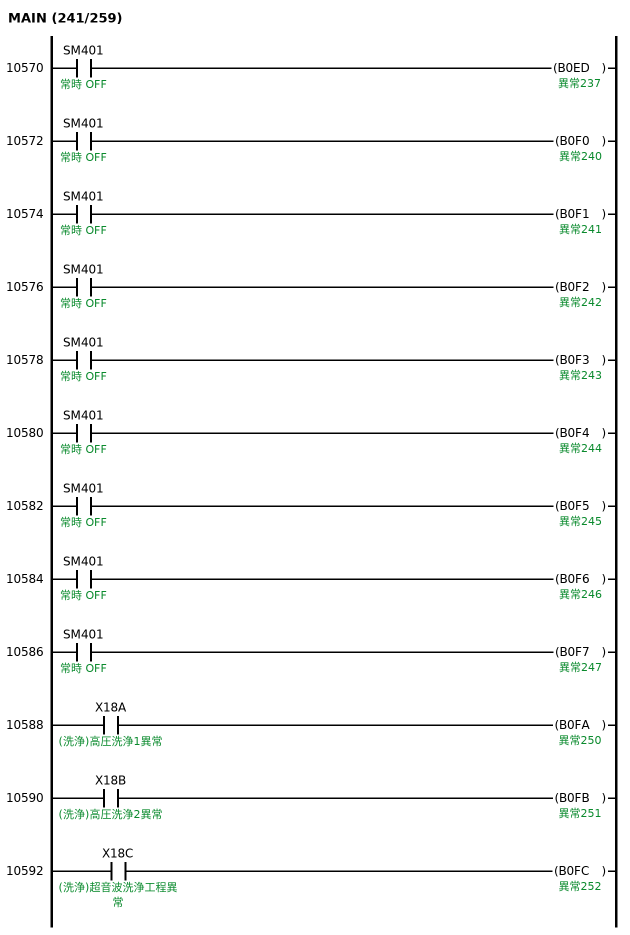
[picture p240: ladder of MAIN, rungs at steps 10570 to 10592]
10570 LD      SM401  ; 常時 OFF
      OUT     B0ED  ; 異常237
10572 LD      SM401  ; 常時 OFF
      OUT     B0F0  ; 異常240
10574 LD      SM401  ; 常時 OFF
      OUT     B0F1  ; 異常241
10576 LD      SM401  ; 常時 OFF
      OUT     B0F2  ; 異常242
10578 LD      SM401  ; 常時 OFF
      OUT     B0F3  ; 異常243
10580 LD      SM401  ; 常時 OFF
      OUT     B0F4  ; 異常244
10582 LD      SM401  ; 常時 OFF
      OUT     B0F5  ; 異常245
10584 LD      SM401  ; 常時 OFF
      OUT     B0F6  ; 異常246
10586 LD      SM401  ; 常時 OFF
      OUT     B0F7  ; 異常247
10588 LD      X18A  ; (洗浄)高圧洗浄1異常
      OUT     B0FA  ; 異常250
10590 LD      X18B  ; (洗浄)高圧洗浄2異常
      OUT     B0FB  ; 異常251
10592 LD      X18C  ; (洗浄)超音波洗浄工程異常
      OUT     B0FC  ; 異常252
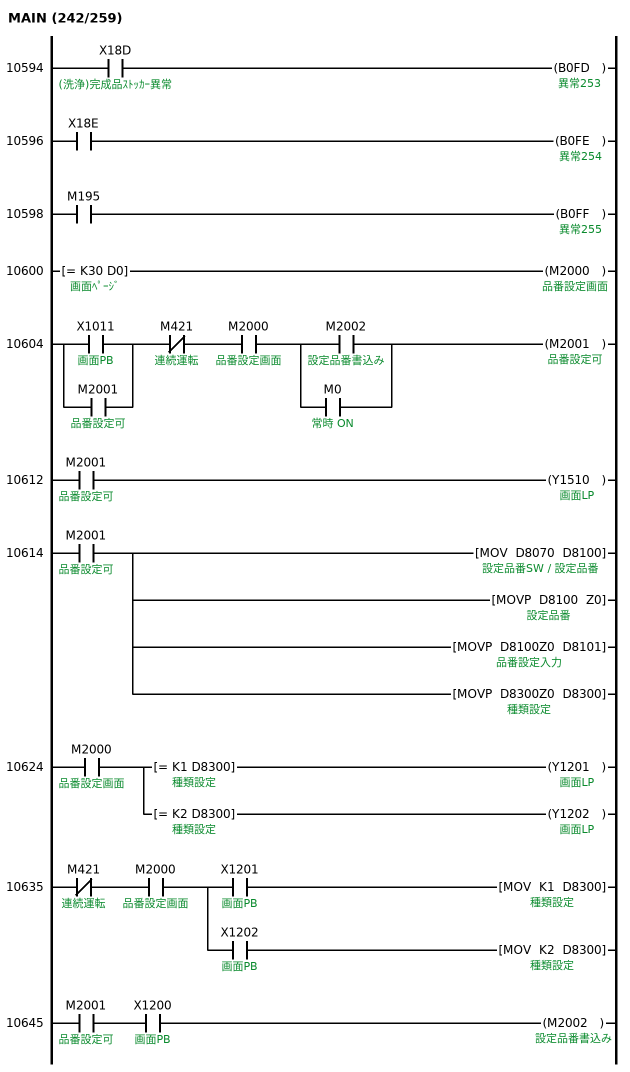
10594 LD      X18D  ; (洗浄)完成品ｽﾄｯｶｰ異常
      OUT     B0FD  ; 異常253
10596 LD      X18E
      OUT     B0FE  ; 異常254
10598 LD      M195
      OUT     B0FF  ; 異常255
10600 LD=     K30 D0  ; 画面ﾍﾟｰｼﾞ
      OUT     M2000  ; 品番設定画面
10604 LD      X1011  ; 画面PB
      OR      M2001  ; 品番設定可
      ANI     M421  ; 連続運転
      AND     M2000  ; 品番設定画面
      LD      M2002  ; 設定品番書込み
      OR      M0  ; 常時 ON
      ANB
      OUT     M2001  ; 品番設定可
10612 LD      M2001  ; 品番設定可
      OUT     Y1510  ; 画面LP
10614 LD      M2001  ; 品番設定可
      MOV     D8070 D8100  ; 設定品番SW / 設定品番
      MOVP    D8100 Z0
      MOVP    D8100Z0 D8101  ; 品番設定入力
      MOVP    D8300Z0 D8300
10624 LD      M2000  ; 品番設定画面
      MPS
      AND=    K1 D8300  ; 種類設定
      OUT     Y1201  ; 画面LP
      MPP
      AND=    K2 D8300  ; 種類設定
      OUT     Y1202  ; 画面LP
10635 LDI     M421  ; 連続運転
      AND     M2000  ; 品番設定画面
      MPS
      AND     X1201  ; 画面PB
      MOV     K1 D8300
      MPP
      AND     X1202  ; 画面PB
      MOV     K2 D8300
10645 LD      M2001  ; 品番設定可
      AND     X1200  ; 画面PB
      OUT     M2002  ; 設定品番書込み
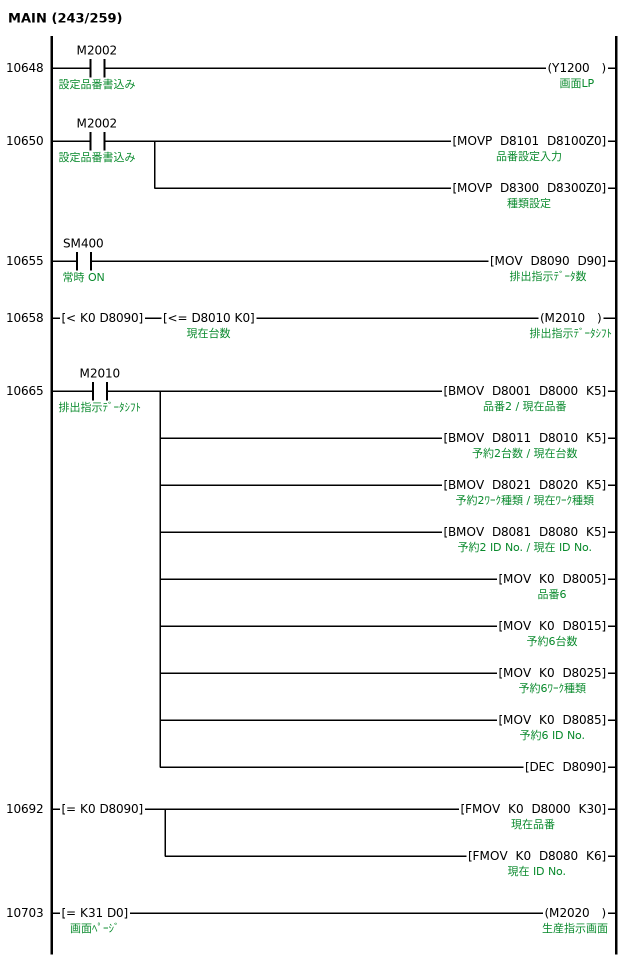
10648 LD      M2002  ; 設定品番書込み
      OUT     Y1200  ; 画面LP
10650 LD      M2002  ; 設定品番書込み
      MOVP    D8101 D8100Z0
      MOVP    D8300 D8300Z0
10655 LD      SM400  ; 常時 ON
      MOV     D8090 D90  ; 排出指示ﾃﾞｰﾀ数
10658 LD<     K0 D8090
      AND<=   D8010 K0  ; 現在台数
      OUT     M2010  ; 排出指示ﾃﾞｰﾀｼﾌﾄ
10665 LD      M2010  ; 排出指示ﾃﾞｰﾀｼﾌﾄ
      BMOV    D8001 D8000 K5  ; 品番2
      BMOV    D8011 D8010 K5  ; 予約2台数
      BMOV    D8021 D8020 K5  ; 予約2ﾜｰｸ種類 / 現在ﾜｰｸ種類
      BMOV    D8081 D8080 K5  ; 予約2 ID No. / 現在 ID No.
      MOV     K0 D8005  ; 品番6
      MOV     K0 D8015  ; 予約6台数
      MOV     K0 D8025  ; 予約6ﾜｰｸ種類
      MOV     K0 D8085  ; 予約6 ID No.
      DEC     D8090
10692 LD=     K0 D8090
      FMOV    K0 D8000 K30
      FMOV    K0 D8080 K6
10703 LD=     K31 D0  ; 画面ﾍﾟｰｼﾞ
      OUT     M2020  ; 生産指示画面
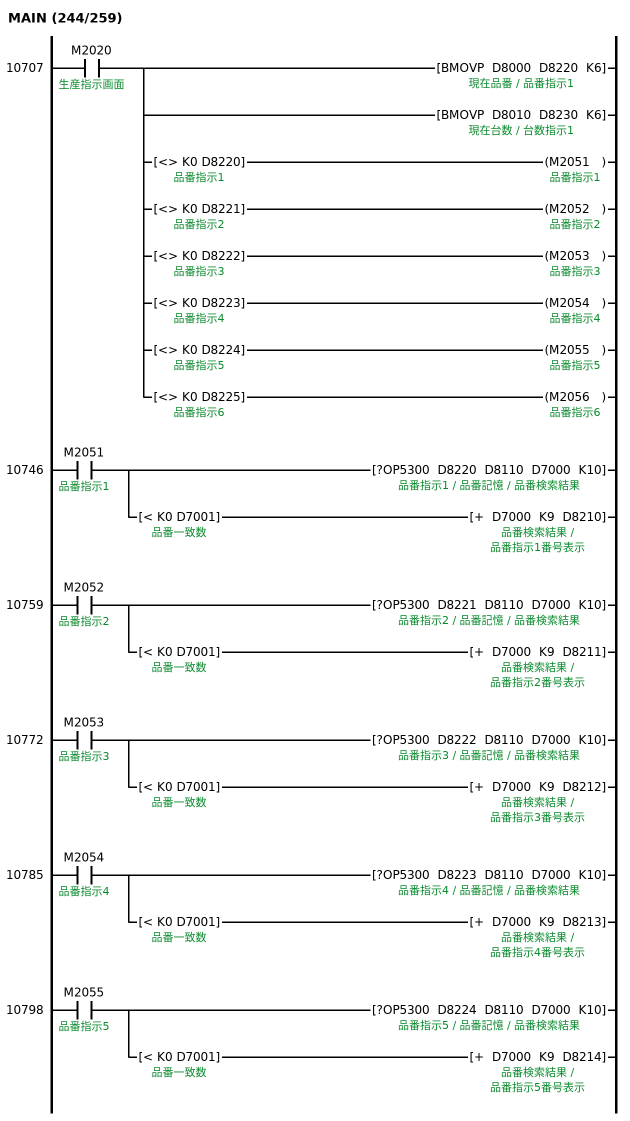
10707 LD      M2020  ; 生産指示画面
      BMOVP   D8000 D8220 K6  ; 品番指示1
      BMOVP   D8010 D8230 K6  ; 台数指示1
      MPS
      AND<>   K0 D8220  ; 品番指示1
      OUT     M2051  ; 品番指示1
      MRD
      AND<>   K0 D8221  ; 品番指示2
      OUT     M2052  ; 品番指示2
      MRD
      AND<>   K0 D8222  ; 品番指示3
      OUT     M2053  ; 品番指示3
      MRD
      AND<>   K0 D8223  ; 品番指示4
      OUT     M2054  ; 品番指示4
      MRD
      AND<>   K0 D8224  ; 品番指示5
      OUT     M2055  ; 品番指示5
      MPP
      AND<>   K0 D8225  ; 品番指示6
      OUT     M2056  ; 品番指示6
10746 LD      M2051  ; 品番指示1
      ?OP5300 D8220 D8110 D7000 K10  ; 品番記憶 / 品番検索結果
      AND<    K0 D7001  ; 品番一致数
      +       D7000 K9 D8210  ; 品番指示1番号表示
10759 LD      M2052  ; 品番指示2
      ?OP5300 D8221 D8110 D7000 K10
      AND<    K0 D7001  ; 品番一致数
      +       D7000 K9 D8211  ; 品番指示2番号表示
10772 LD      M2053  ; 品番指示3
      ?OP5300 D8222 D8110 D7000 K10
      AND<    K0 D7001  ; 品番一致数
      +       D7000 K9 D8212  ; 品番指示3番号表示
10785 LD      M2054  ; 品番指示4
      ?OP5300 D8223 D8110 D7000 K10
      AND<    K0 D7001  ; 品番一致数
      +       D7000 K9 D8213  ; 品番指示4番号表示
10798 LD      M2055  ; 品番指示5
      ?OP5300 D8224 D8110 D7000 K10
      AND<    K0 D7001  ; 品番一致数
      +       D7000 K9 D8214  ; 品番指示5番号表示
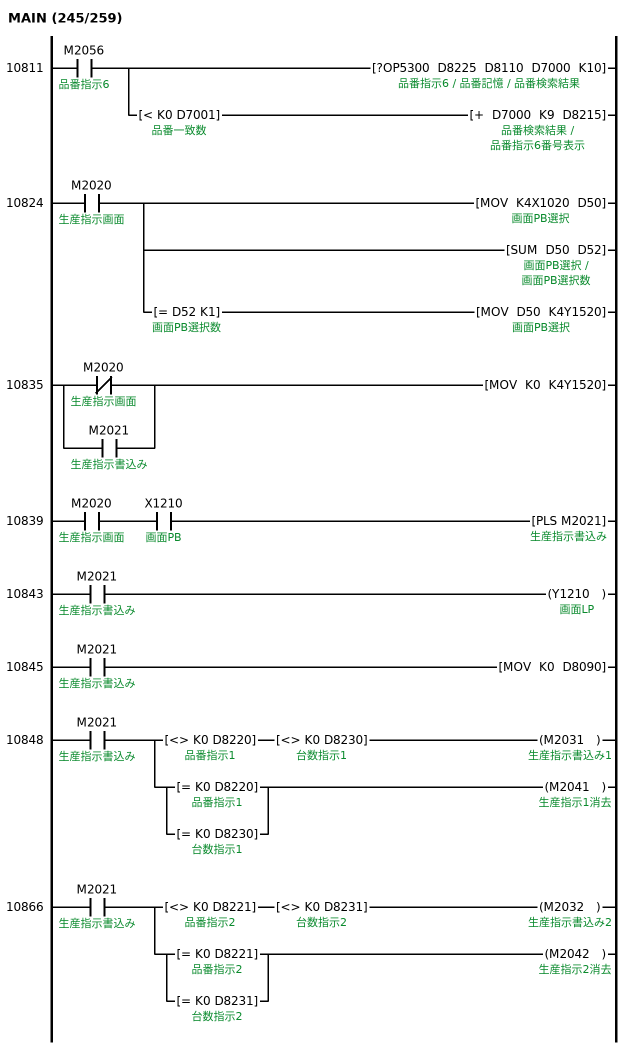
10811 LD      M2056  ; 品番指示6
      ?OP5300 D8225 D8110 D7000 K10
      AND<    K0 D7001  ; 品番一致数
      +       D7000 K9 D8215  ; 品番指示6番号表示
10824 LD      M2020  ; 生産指示画面
      MOV     K4X1020 D50  ; 画面PB
      SUM     D50 D52
      AND=    D52 K1  ; 画面PB選択数
      MOV     D50 K4Y1520  ; 画面LP
10835 LDI     M2020  ; 生産指示画面
      OR      M2021  ; 生産指示書込み
      MOV     K0 K4Y1520
10839 LD      M2020  ; 生産指示画面
      AND     X1210  ; 画面PB
      PLS     M2021  ; 生産指示書込み
10843 LD      M2021  ; 生産指示書込み
      OUT     Y1210  ; 画面LP
10845 LD      M2021  ; 生産指示書込み
      MOV     K0 D8090
10848 LD      M2021  ; 生産指示書込み
      MPS
      AND<>   K0 D8220  ; 品番指示1
      AND<>   K0 D8230  ; 台数指示1
      OUT     M2031  ; 生産指示書込み1
      MPP
      LD=     K0 D8220  ; 品番指示1
      OR=     K0 D8230  ; 台数指示1
      ANB
      OUT     M2041  ; 生産指示1消去
10866 LD      M2021  ; 生産指示書込み
      MPS
      AND<>   K0 D8221  ; 品番指示2
      AND<>   K0 D8231  ; 台数指示2
      OUT     M2032  ; 生産指示書込み2
      MPP
      LD=     K0 D8221  ; 品番指示2
      OR=     K0 D8231  ; 台数指示2
      ANB
      OUT     M2042  ; 生産指示2消去
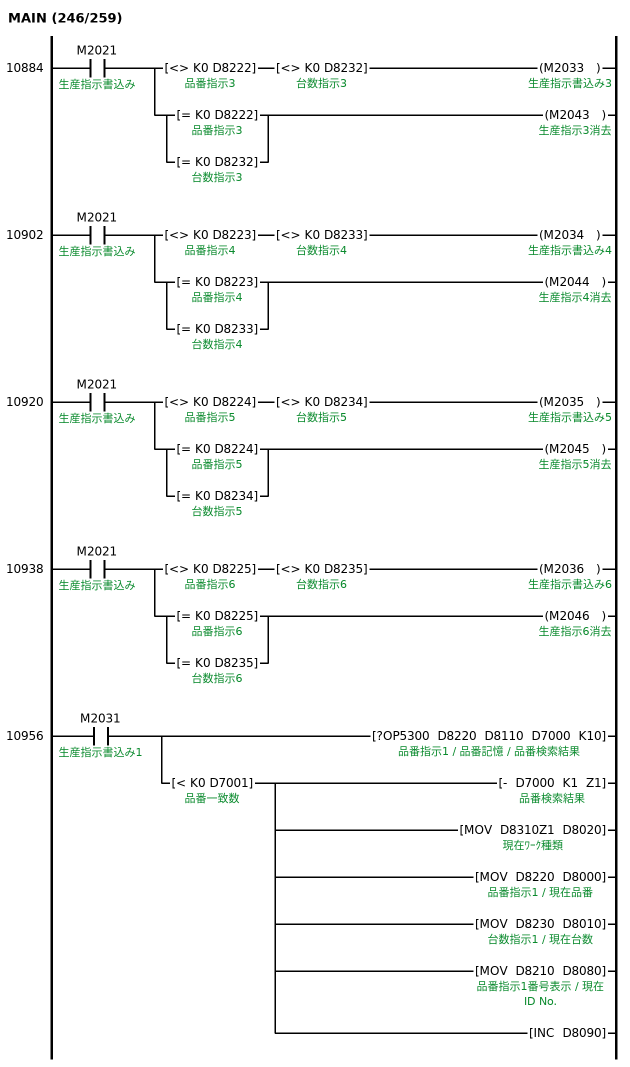
10884 LD      M2021  ; 生産指示書込み
      MPS
      AND<>   K0 D8222  ; 品番指示3
      AND<>   K0 D8232  ; 台数指示3
      OUT     M2033  ; 生産指示書込み3
      MPP
      LD=     K0 D8222  ; 品番指示3
      OR=     K0 D8232  ; 台数指示3
      ANB
      OUT     M2043  ; 生産指示3消去
10902 LD      M2021  ; 生産指示書込み
      MPS
      AND<>   K0 D8223  ; 品番指示4
      AND<>   K0 D8233  ; 台数指示4
      OUT     M2034  ; 生産指示書込み4
      MPP
      LD=     K0 D8223  ; 品番指示4
      OR=     K0 D8233  ; 台数指示4
      ANB
      OUT     M2044  ; 生産指示4消去
10920 LD      M2021  ; 生産指示書込み
      MPS
      AND<>   K0 D8224  ; 品番指示5
      AND<>   K0 D8234  ; 台数指示5
      OUT     M2035  ; 生産指示書込み5
      MPP
      LD=     K0 D8224  ; 品番指示5
      OR=     K0 D8234  ; 台数指示5
      ANB
      OUT     M2045  ; 生産指示5消去
10938 LD      M2021  ; 生産指示書込み
      MPS
      AND<>   K0 D8225  ; 品番指示6
      AND<>   K0 D8235  ; 台数指示6
      OUT     M2036  ; 生産指示書込み6
      MPP
      LD=     K0 D8225  ; 品番指示6
      OR=     K0 D8235  ; 台数指示6
      ANB
      OUT     M2046  ; 生産指示6消去
10956 LD      M2031  ; 生産指示書込み1
      ?OP5300 D8220 D8110 D7000 K10
      AND<    K0 D7001  ; 品番一致数
      -       D7000 K1 Z1
      MOV     D8310Z1 D8020
      MOV     D8220 D8000
      MOV     D8230 D8010
      MOV     D8210 D8080
      INC     D8090
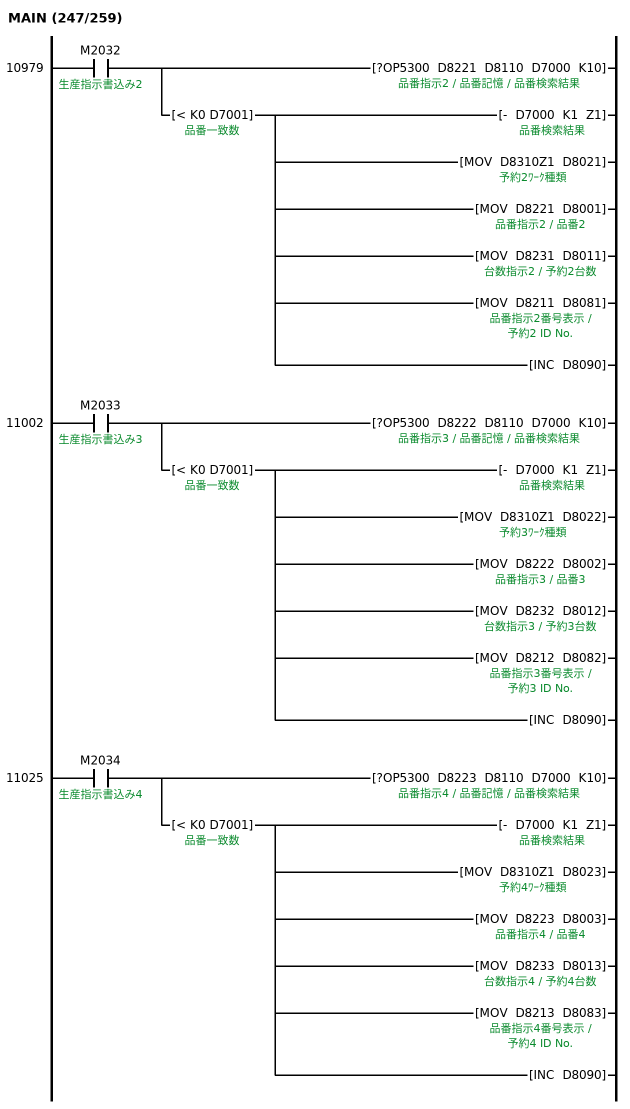
10979 LD      M2032  ; 生産指示書込み2
      ?OP5300 D8221 D8110 D7000 K10
      AND<    K0 D7001  ; 品番一致数
      -       D7000 K1 Z1
      MOV     D8310Z1 D8021
      MOV     D8221 D8001
      MOV     D8231 D8011
      MOV     D8211 D8081
      INC     D8090
11002 LD      M2033  ; 生産指示書込み3
      ?OP5300 D8222 D8110 D7000 K10
      AND<    K0 D7001  ; 品番一致数
      -       D7000 K1 Z1
      MOV     D8310Z1 D8022  ; 予約3ﾜｰｸ種類
      MOV     D8222 D8002  ; 品番3
      MOV     D8232 D8012  ; 予約3台数
      MOV     D8212 D8082  ; 予約3 ID No.
      INC     D8090
11025 LD      M2034  ; 生産指示書込み4
      ?OP5300 D8223 D8110 D7000 K10
      AND<    K0 D7001  ; 品番一致数
      -       D7000 K1 Z1
      MOV     D8310Z1 D8023  ; 予約4ﾜｰｸ種類
      MOV     D8223 D8003  ; 品番4
      MOV     D8233 D8013  ; 予約4台数
      MOV     D8213 D8083  ; 予約4 ID No.
      INC     D8090
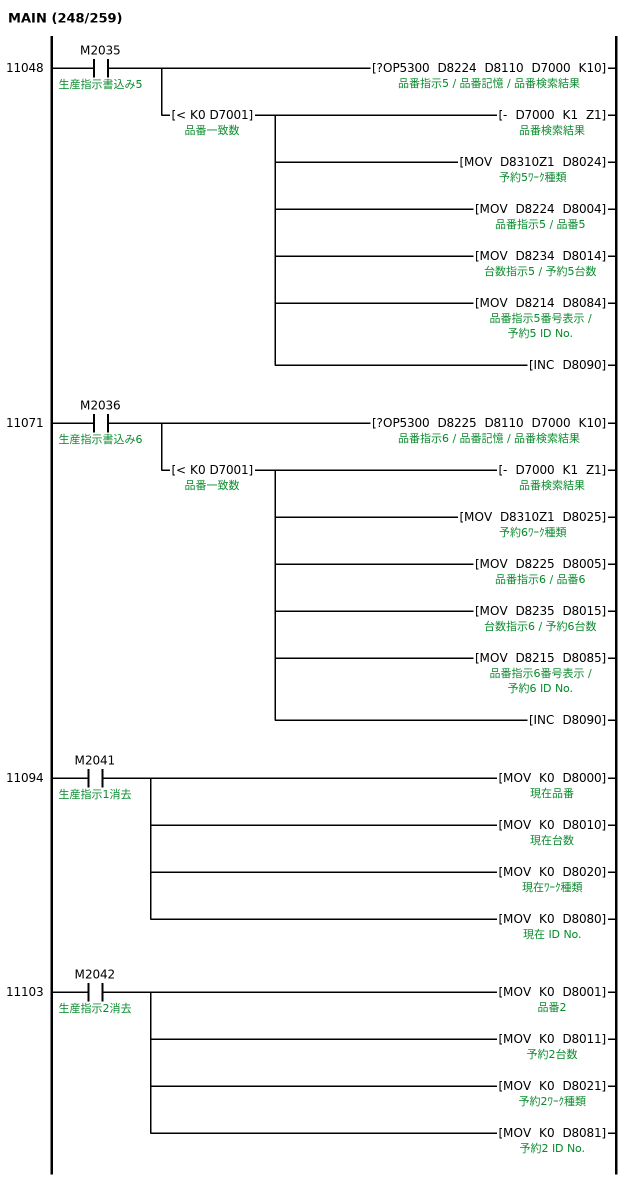
11048 LD      M2035  ; 生産指示書込み5
      ?OP5300 D8224 D8110 D7000 K10
      AND<    K0 D7001  ; 品番一致数
      -       D7000 K1 Z1
      MOV     D8310Z1 D8024  ; 予約5ﾜｰｸ種類
      MOV     D8224 D8004  ; 品番5
      MOV     D8234 D8014  ; 予約5台数
      MOV     D8214 D8084  ; 予約5 ID No.
      INC     D8090
11071 LD      M2036  ; 生産指示書込み6
      ?OP5300 D8225 D8110 D7000 K10
      AND<    K0 D7001  ; 品番一致数
      -       D7000 K1 Z1
      MOV     D8310Z1 D8025
      MOV     D8225 D8005
      MOV     D8235 D8015
      MOV     D8215 D8085
      INC     D8090
11094 LD      M2041  ; 生産指示1消去
      MOV     K0 D8000
      MOV     K0 D8010
      MOV     K0 D8020
      MOV     K0 D8080
11103 LD      M2042  ; 生産指示2消去
      MOV     K0 D8001
      MOV     K0 D8011
      MOV     K0 D8021
      MOV     K0 D8081
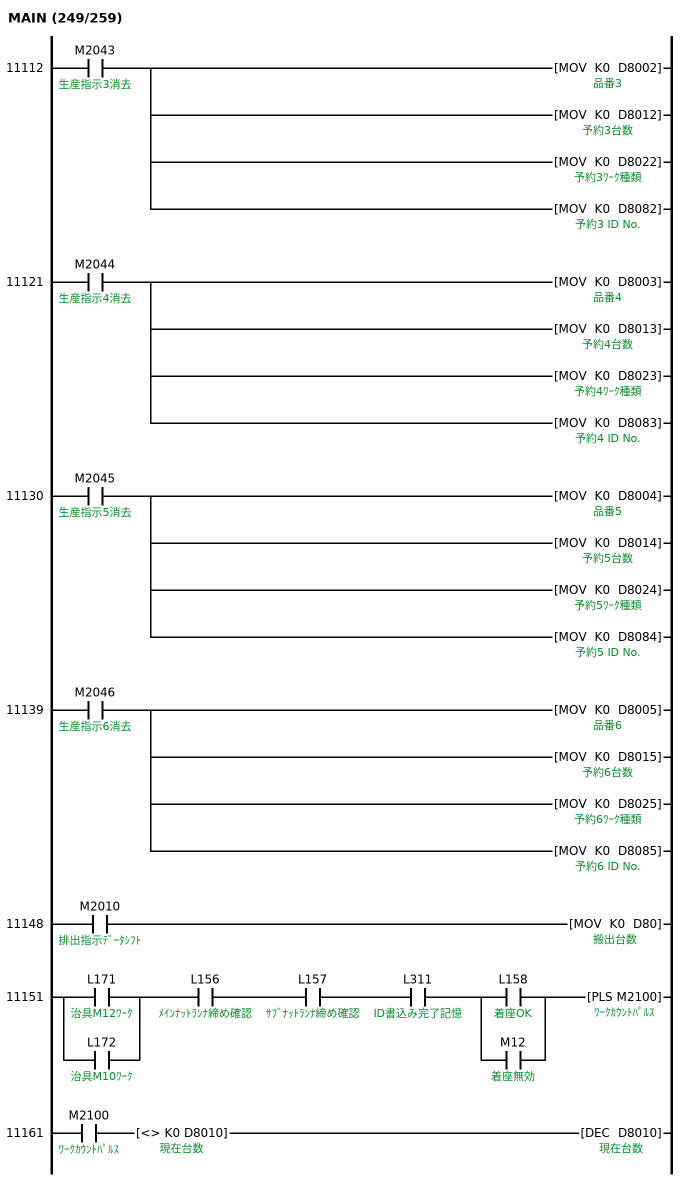
11112 LD      M2043  ; 生産指示3消去
      MOV     K0 D8002
      MOV     K0 D8012
      MOV     K0 D8022
      MOV     K0 D8082
11121 LD      M2044  ; 生産指示4消去
      MOV     K0 D8003
      MOV     K0 D8013
      MOV     K0 D8023
      MOV     K0 D8083
11130 LD      M2045  ; 生産指示5消去
      MOV     K0 D8004
      MOV     K0 D8014
      MOV     K0 D8024
      MOV     K0 D8084
11139 LD      M2046  ; 生産指示6消去
      MOV     K0 D8005
      MOV     K0 D8015
      MOV     K0 D8025
      MOV     K0 D8085
11148 LD      M2010  ; 排出指示ﾃﾞｰﾀｼﾌﾄ
      MOV     K0 D80  ; 搬出台数
11151 LD      L171  ; 治具M12ﾜｰｸ
      OR      L172  ; 治具M10ﾜｰｸ
      AND     L156  ; ﾒｲﾝﾅｯﾄﾗﾝﾅ締め確認
      AND     L157  ; ｻﾌﾞﾅｯﾄﾗﾝﾅ締め確認
      AND     L311  ; ID書込み完了記憶
      LD      L158  ; 着座OK
      OR      M12  ; 着座無効
      ANB
      PLS     M2100  ; ﾜｰｸｶｳﾝﾄﾊﾟﾙｽ
11161 LD      M2100  ; ﾜｰｸｶｳﾝﾄﾊﾟﾙｽ
      AND<>   K0 D8010  ; 現在台数
      DEC     D8010
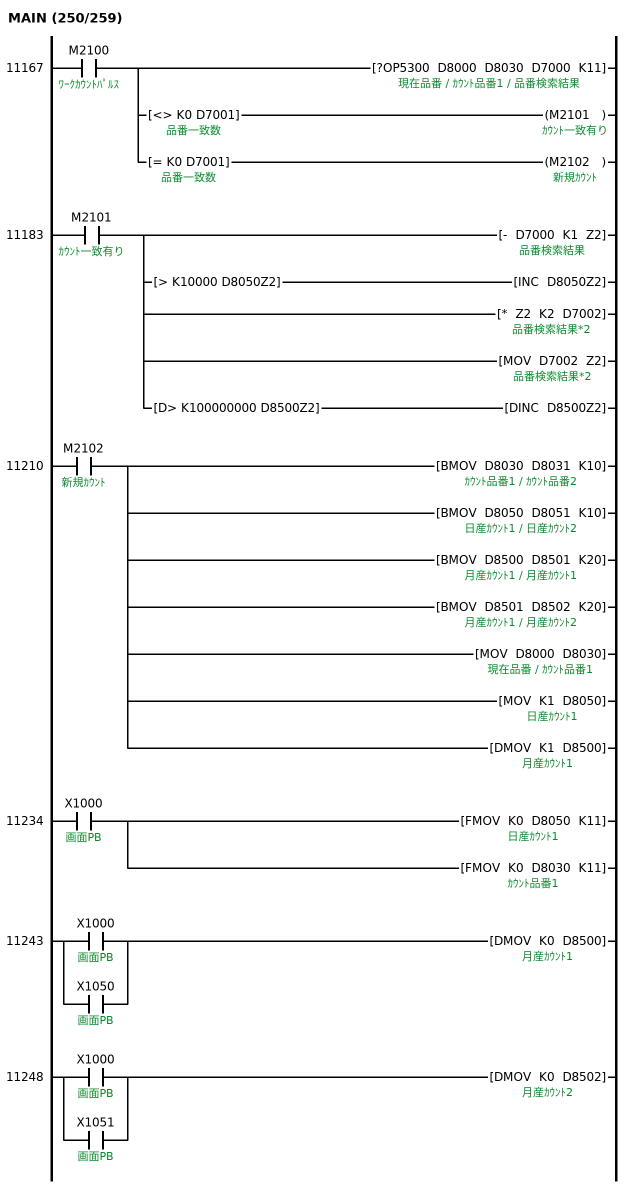
11167 LD      M2100  ; ﾜｰｸｶｳﾝﾄﾊﾟﾙｽ
      ?OP5300 D8000 D8030 D7000 K11  ; ｶｳﾝﾄ品番1
      MPS
      AND<>   K0 D7001  ; 品番一致数
      OUT     M2101  ; ｶｳﾝﾄ一致有り
      MPP
      AND=    K0 D7001  ; 品番一致数
      OUT     M2102  ; 新規ｶｳﾝﾄ
11183 LD      M2101  ; ｶｳﾝﾄ一致有り
      -       D7000 K1 Z2
      MPS
      AND>    K10000 D8050Z2
      INC     D8050Z2
      MPP
      *       Z2 K2 D7002  ; 品番検索結果*2
      MOV     D7002 Z2
      ANDD>   K100000000 D8500Z2
      DINC    D8500Z2
11210 LD      M2102  ; 新規ｶｳﾝﾄ
      BMOV    D8030 D8031 K10  ; ｶｳﾝﾄ品番2
      BMOV    D8050 D8051 K10  ; 日産ｶｳﾝﾄ1 / 日産ｶｳﾝﾄ2
      BMOV    D8500 D8501 K20  ; 月産ｶｳﾝﾄ1 / 月産ｶｳﾝﾄ1
      BMOV    D8501 D8502 K20  ; 月産ｶｳﾝﾄ2
      MOV     D8000 D8030
      MOV     K1 D8050
      DMOV    K1 D8500
11234 LD      X1000  ; 画面PB
      FMOV    K0 D8050 K11
      FMOV    K0 D8030 K11
11243 LD      X1000  ; 画面PB
      OR      X1050  ; 画面PB
      DMOV    K0 D8500
11248 LD      X1000  ; 画面PB
      OR      X1051  ; 画面PB
      DMOV    K0 D8502
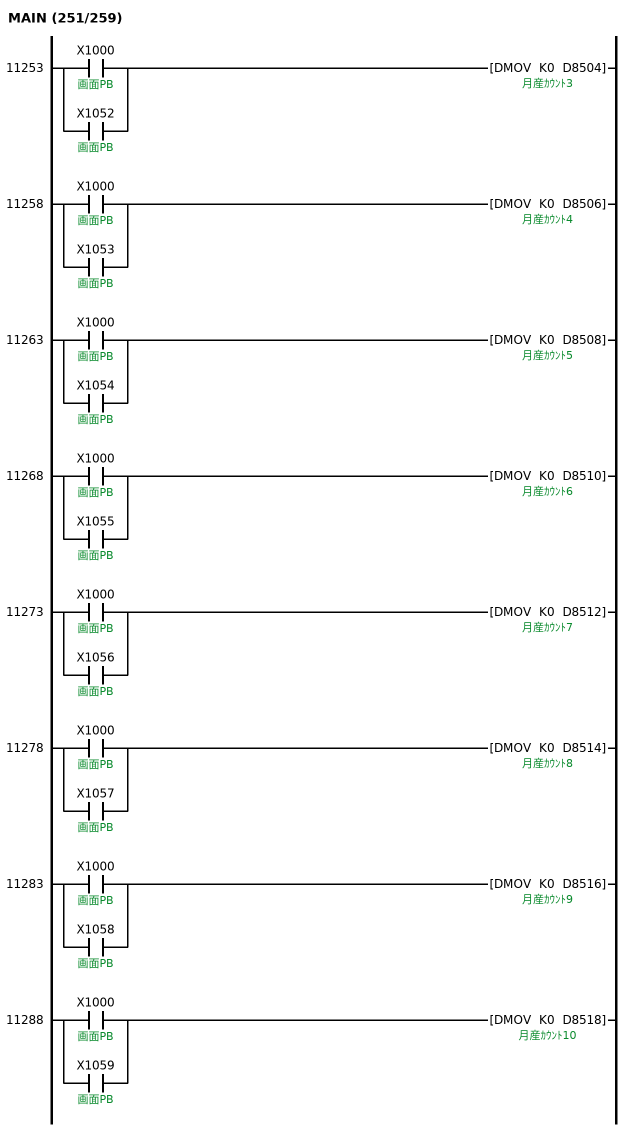
11253 LD      X1000  ; 画面PB
      OR      X1052  ; 画面PB
      DMOV    K0 D8504  ; 月産ｶｳﾝﾄ3
11258 LD      X1000  ; 画面PB
      OR      X1053  ; 画面PB
      DMOV    K0 D8506  ; 月産ｶｳﾝﾄ4
11263 LD      X1000  ; 画面PB
      OR      X1054  ; 画面PB
      DMOV    K0 D8508  ; 月産ｶｳﾝﾄ5
11268 LD      X1000  ; 画面PB
      OR      X1055  ; 画面PB
      DMOV    K0 D8510  ; 月産ｶｳﾝﾄ6
11273 LD      X1000  ; 画面PB
      OR      X1056  ; 画面PB
      DMOV    K0 D8512  ; 月産ｶｳﾝﾄ7
11278 LD      X1000  ; 画面PB
      OR      X1057  ; 画面PB
      DMOV    K0 D8514  ; 月産ｶｳﾝﾄ8
11283 LD      X1000  ; 画面PB
      OR      X1058  ; 画面PB
      DMOV    K0 D8516  ; 月産ｶｳﾝﾄ9
11288 LD      X1000  ; 画面PB
      OR      X1059  ; 画面PB
      DMOV    K0 D8518  ; 月産ｶｳﾝﾄ10
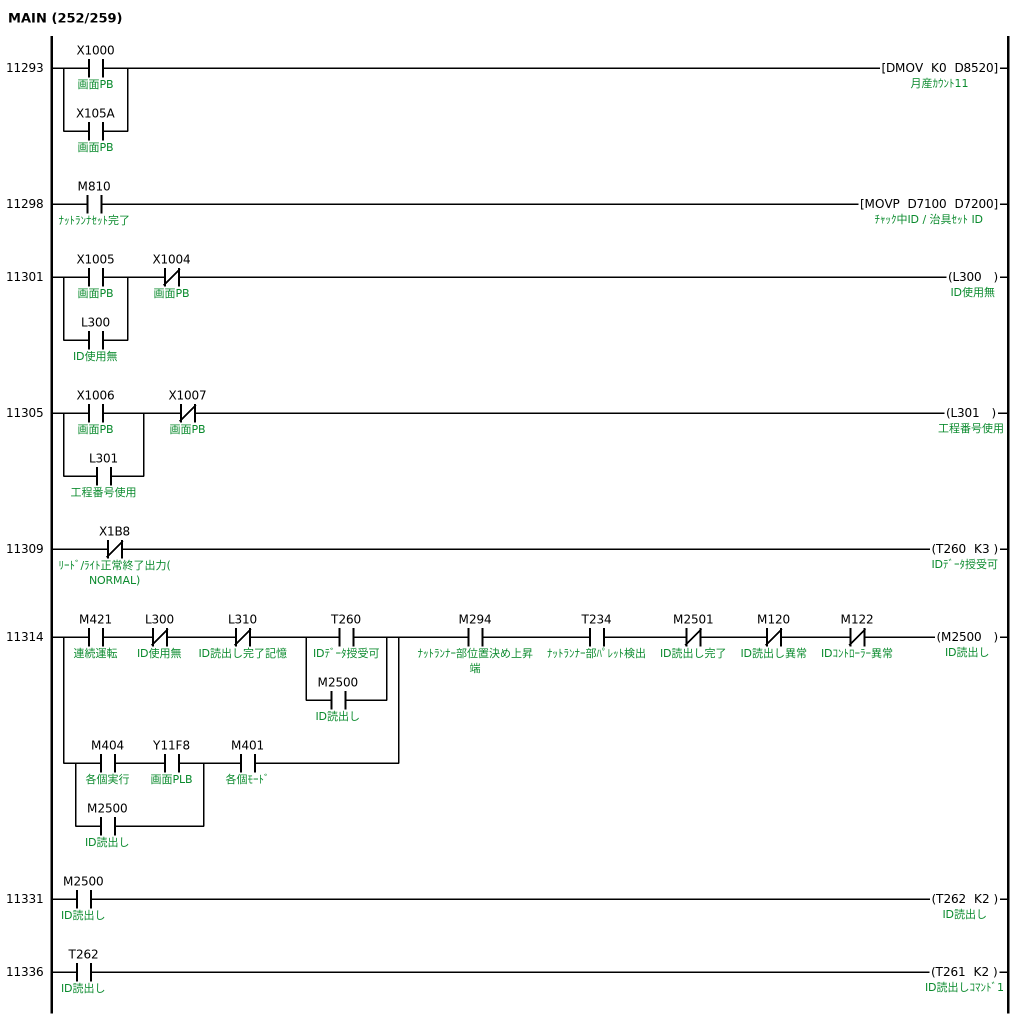
11293 LD      X1000  ; 画面PB
      OR      X105A  ; 画面PB
      DMOV    K0 D8520  ; 月産ｶｳﾝﾄ11
11298 LD      M810  ; ﾅｯﾄﾗﾝﾅｾｯﾄ完了
      MOVP    D7100 D7200  ; 治具ｾｯﾄ ID
11301 LD      X1005  ; 画面PB
      OR      L300  ; ID使用無
      ANI     X1004  ; 画面PB
      OUT     L300  ; ID使用無
11305 LD      X1006  ; 画面PB
      OR      L301  ; 工程番号使用
      ANI     X1007  ; 画面PB
      OUT     L301  ; 工程番号使用
11309 LDI     X1B8  ; ﾘｰﾄﾞ/ﾗｲﾄ正常終了出力(NORMAL)
      OUT     T260 K3  ; IDﾃﾞｰﾀ授受可
11314 LD      M421  ; 連続運転
      ANI     L300  ; ID使用無
      ANI     L310  ; ID読出し完了記憶
      LD      T260  ; IDﾃﾞｰﾀ授受可
      OR      M2500  ; ID読出し
      ANB
      LD      M404  ; 各個実行
      AND     Y11F8  ; 画面PLB
      OR      M2500  ; ID読出し
      AND     M401  ; 各個ﾓｰﾄﾞ
      ORB
      AND     M294  ; ﾅｯﾄﾗﾝﾅｰ部位置決め上昇端
      AND     T234  ; ﾅｯﾄﾗﾝﾅｰ部ﾊﾟﾚｯﾄ検出
      ANI     M2501  ; ID読出し完了
      ANI     M120  ; ID読出し異常
      ANI     M122  ; IDｺﾝﾄﾛｰﾗｰ異常
      OUT     M2500  ; ID読出し
11331 LD      M2500  ; ID読出し
      OUT     T262 K2  ; ID読出し
11336 LD      T262  ; ID読出し
      OUT     T261 K2  ; ID読出しｺﾏﾝﾄﾞ1
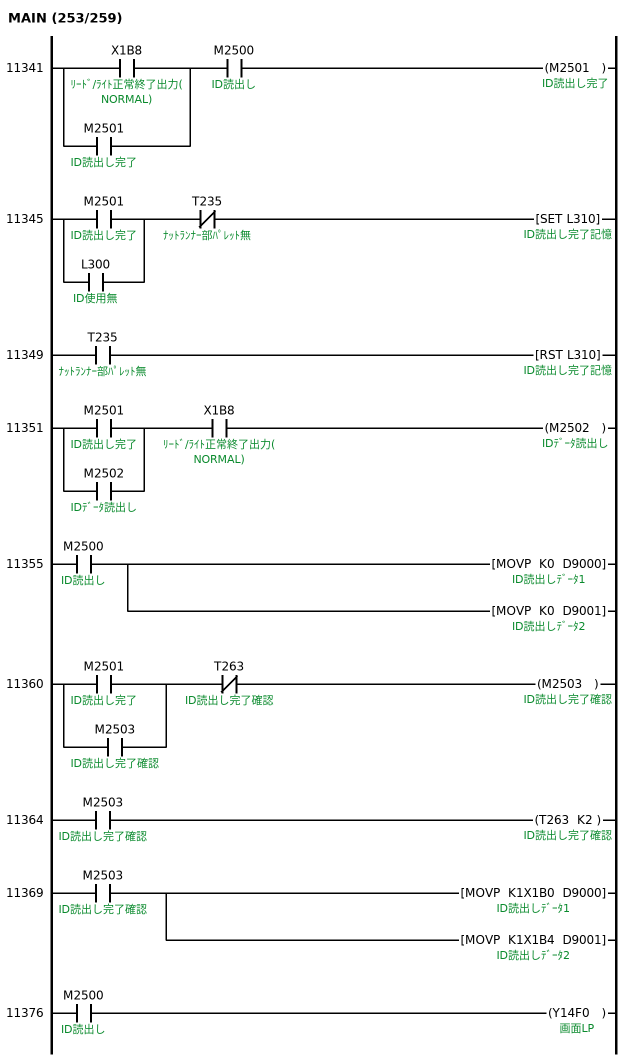
11341 LD      X1B8  ; ﾘｰﾄﾞ/ﾗｲﾄ正常終了出力(NORMAL)
      OR      M2501  ; ID読出し完了
      AND     M2500  ; ID読出し
      OUT     M2501  ; ID読出し完了
11345 LD      M2501  ; ID読出し完了
      OR      L300  ; ID使用無
      ANI     T235  ; ﾅｯﾄﾗﾝﾅｰ部ﾊﾟﾚｯﾄ無
      SET     L310  ; ID読出し完了記憶
11349 LD      T235  ; ﾅｯﾄﾗﾝﾅｰ部ﾊﾟﾚｯﾄ無
      RST     L310  ; ID読出し完了記憶
11351 LD      M2501  ; ID読出し完了
      OR      M2502  ; IDﾃﾞｰﾀ読出し
      AND     X1B8  ; ﾘｰﾄﾞ/ﾗｲﾄ正常終了出力(NORMAL)
      OUT     M2502  ; IDﾃﾞｰﾀ読出し
11355 LD      M2500  ; ID読出し
      MOVP    K0 D9000  ; ID読出しﾃﾞｰﾀ1
      MOVP    K0 D9001  ; ID読出しﾃﾞｰﾀ2
11360 LD      M2501  ; ID読出し完了
      OR      M2503  ; ID読出し完了確認
      ANI     T263  ; ID読出し完了確認
      OUT     M2503  ; ID読出し完了確認
11364 LD      M2503  ; ID読出し完了確認
      OUT     T263 K2  ; ID読出し完了確認
11369 LD      M2503  ; ID読出し完了確認
      MOVP    K1X1B0 D9000  ; ﾘｰﾄﾞﾃﾞｰﾀ出力ﾋﾞｯﾄ0(OD0)
      MOVP    K1X1B4 D9001  ; ﾘｰﾄﾞﾃﾞｰﾀ出力ﾋﾞｯﾄ4(OD4)
11376 LD      M2500  ; ID読出し
      OUT     Y14F0  ; 画面LP
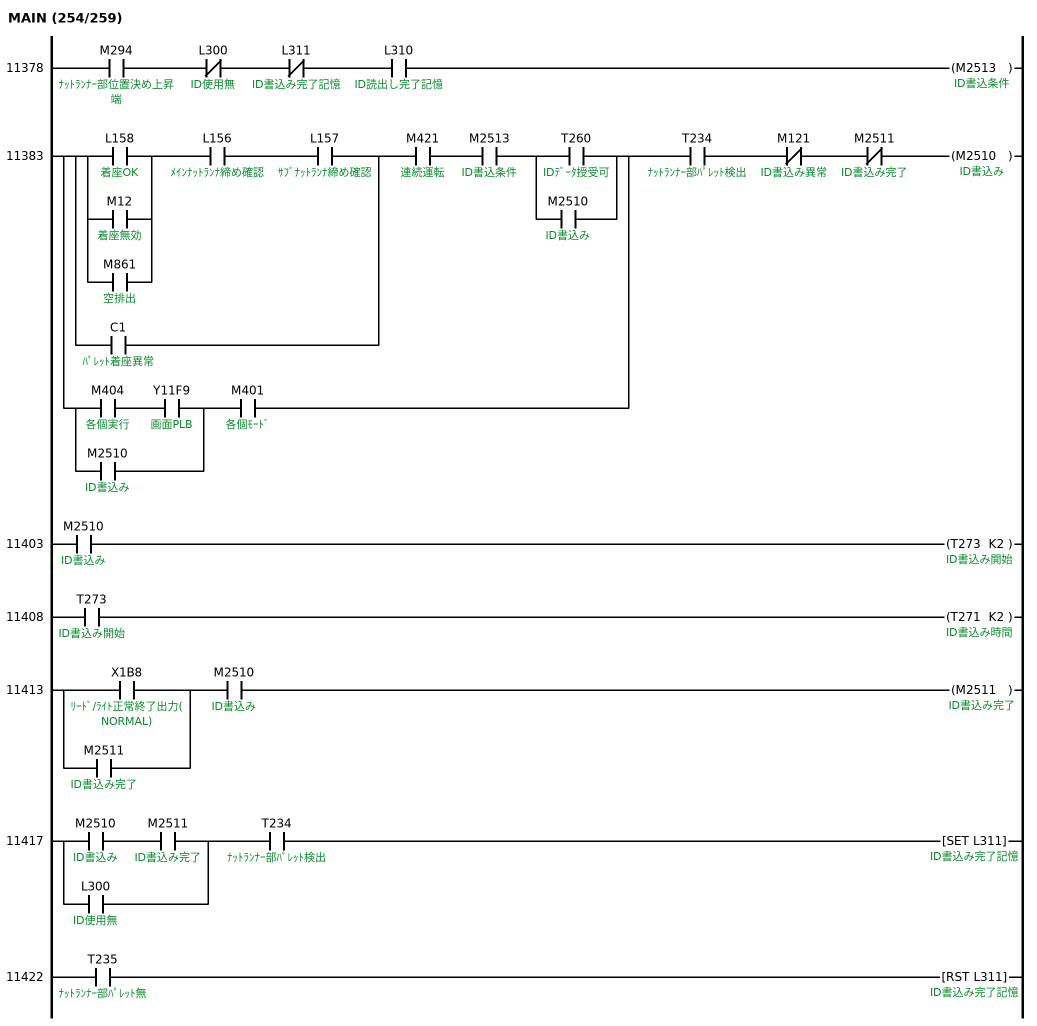
11378 LD      M294  ; ﾅｯﾄﾗﾝﾅｰ部位置決め上昇端
      ANI     L300  ; ID使用無
      ANI     L311  ; ID書込み完了記憶
      AND     L310  ; ID読出し完了記憶
      OUT     M2513  ; ID書込条件
11383 LD      L158  ; 着座OK
      OR      M12  ; 着座無効
      OR      M861  ; 空排出
      AND     L156  ; ﾒｲﾝﾅｯﾄﾗﾝﾅ締め確認
      AND     L157  ; ｻﾌﾞﾅｯﾄﾗﾝﾅ締め確認
      OR      C1  ; ﾊﾟﾚｯﾄ着座異常
      AND     M421  ; 連続運転
      AND     M2513  ; ID書込条件
      LD      T260  ; IDﾃﾞｰﾀ授受可
      OR      M2510  ; ID書込み
      ANB
      LD      M404  ; 各個実行
      AND     Y11F9  ; 画面PLB
      OR      M2510  ; ID書込み
      AND     M401  ; 各個ﾓｰﾄﾞ
      ORB
      AND     T234  ; ﾅｯﾄﾗﾝﾅｰ部ﾊﾟﾚｯﾄ検出
      ANI     M121  ; ID書込み異常
      ANI     M2511  ; ID書込み完了
      OUT     M2510  ; ID書込み
11403 LD      M2510  ; ID書込み
      OUT     T273 K2  ; ID書込み開始
11408 LD      T273  ; ID書込み開始
      OUT     T271 K2  ; ID書込み時間
11413 LD      X1B8  ; ﾘｰﾄﾞ/ﾗｲﾄ正常終了出力(NORMAL)
      OR      M2511  ; ID書込み完了
      AND     M2510  ; ID書込み
      OUT     M2511  ; ID書込み完了
11417 LD      M2510  ; ID書込み
      AND     M2511  ; ID書込み完了
      OR      L300  ; ID使用無
      AND     T234  ; ﾅｯﾄﾗﾝﾅｰ部ﾊﾟﾚｯﾄ検出
      SET     L311  ; ID書込み完了記憶
11422 LD      T235  ; ﾅｯﾄﾗﾝﾅｰ部ﾊﾟﾚｯﾄ無
      RST     L311  ; ID書込み完了記憶
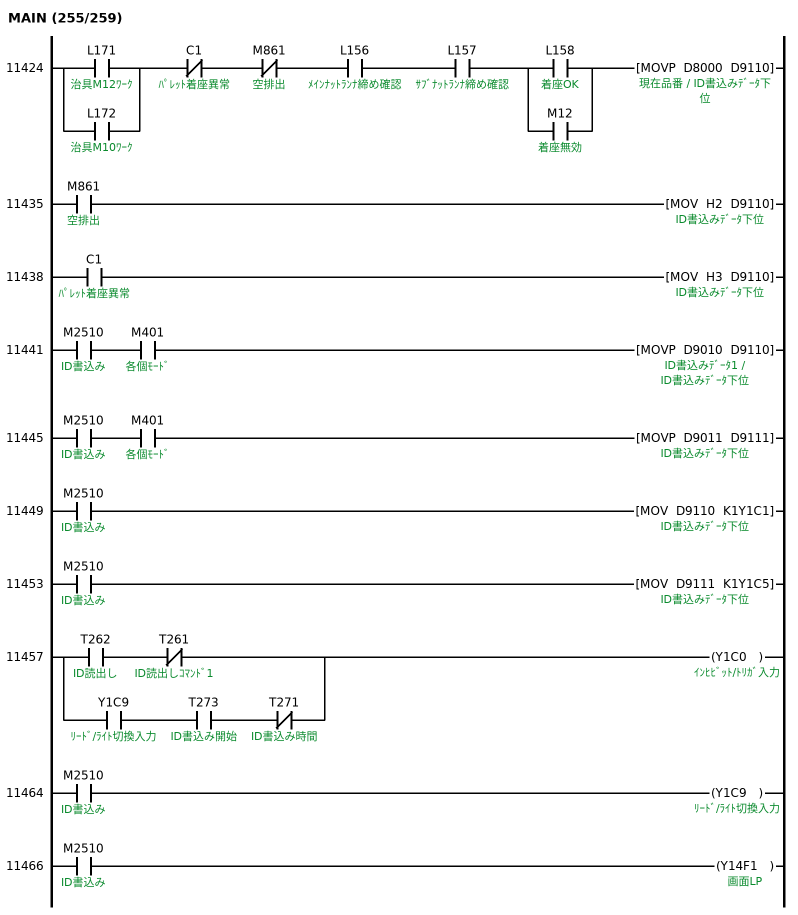
11424 LD      L171  ; 治具M12ﾜｰｸ
      OR      L172  ; 治具M10ﾜｰｸ
      ANI     C1  ; ﾊﾟﾚｯﾄ着座異常
      ANI     M861  ; 空排出
      AND     L156  ; ﾒｲﾝﾅｯﾄﾗﾝﾅ締め確認
      AND     L157  ; ｻﾌﾞﾅｯﾄﾗﾝﾅ締め確認
      LD      L158  ; 着座OK
      OR      M12  ; 着座無効
      ANB
      MOVP    D8000 D9110  ; ID書込みﾃﾞｰﾀ下位
11435 LD      M861  ; 空排出
      MOV     H2 D9110
11438 LD      C1  ; ﾊﾟﾚｯﾄ着座異常
      MOV     H3 D9110
11441 LD      M2510  ; ID書込み
      AND     M401  ; 各個ﾓｰﾄﾞ
      MOVP    D9010 D9110  ; ID書込みﾃﾞｰﾀ1
11445 LD      M2510  ; ID書込み
      AND     M401  ; 各個ﾓｰﾄﾞ
      MOVP    D9011 D9111  ; ID書込みﾃﾞｰﾀ下位
11449 LD      M2510  ; ID書込み
      MOV     D9110 K1Y1C1  ; ﾗｲﾄﾃﾞｰﾀ入力ﾋﾞｯﾄ 0
11453 LD      M2510  ; ID書込み
      MOV     D9111 K1Y1C5  ; ﾗｲﾄﾃﾞｰﾀ入力ﾋﾞｯﾄ 4
11457 LD      T262  ; ID読出し
      ANI     T261  ; ID読出しｺﾏﾝﾄﾞ1
      LD      Y1C9  ; ﾘｰﾄﾞ/ﾗｲﾄ切換入力
      AND     T273  ; ID書込み開始
      ANI     T271  ; ID書込み時間
      ORB
      OUT     Y1C0  ; ｲﾝﾋﾋﾞｯﾄ/ﾄﾘｶﾞ入力
11464 LD      M2510  ; ID書込み
      OUT     Y1C9  ; ﾘｰﾄﾞ/ﾗｲﾄ切換入力
11466 LD      M2510  ; ID書込み
      OUT     Y14F1  ; 画面LP
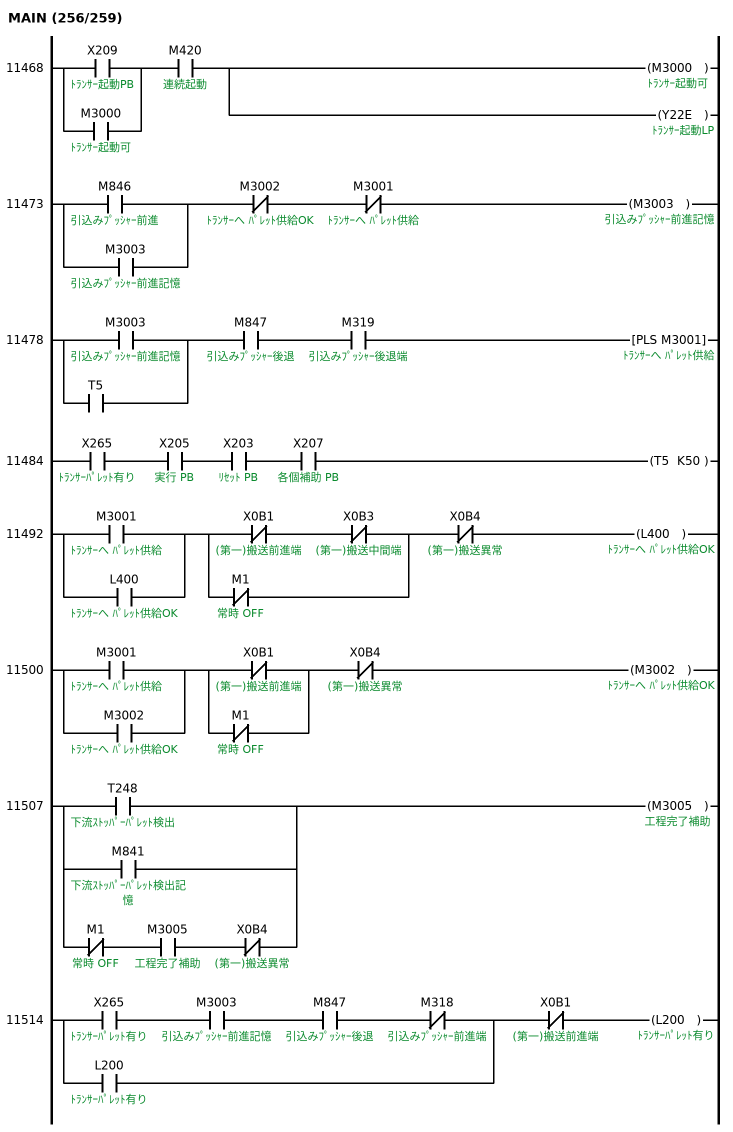
11468 LD      X209  ; ﾄﾗﾝｻｰ起動PB
      OR      M3000  ; ﾄﾗﾝｻｰ起動可
      AND     M420  ; 連続起動
      OUT     M3000  ; ﾄﾗﾝｻｰ起動可
      OUT     Y22E  ; ﾄﾗﾝｻｰ起動LP
11473 LD      M846  ; 引込みﾌﾟｯｼｬｰ前進
      OR      M3003  ; 引込みﾌﾟｯｼｬｰ前進記憶
      ANI     M3002  ; ﾄﾗﾝｻｰへ ﾊﾟﾚｯﾄ供給OK
      ANI     M3001  ; ﾄﾗﾝｻｰへ ﾊﾟﾚｯﾄ供給
      OUT     M3003  ; 引込みﾌﾟｯｼｬｰ前進記憶
11478 LD      M3003  ; 引込みﾌﾟｯｼｬｰ前進記憶
      OR      T5
      AND     M847  ; 引込みﾌﾟｯｼｬｰ後退
      AND     M319  ; 引込みﾌﾟｯｼｬｰ後退端
      PLS     M3001  ; ﾄﾗﾝｻｰへ ﾊﾟﾚｯﾄ供給
11484 LD      X265  ; ﾄﾗﾝｻｰﾊﾟﾚｯﾄ有り
      AND     X205  ; 実行 PB
      AND     X203  ; ﾘｾｯﾄ PB
      AND     X207  ; 各個補助 PB
      OUT     T5 K50
11492 LD      M3001  ; ﾄﾗﾝｻｰへ ﾊﾟﾚｯﾄ供給
      OR      L400  ; ﾄﾗﾝｻｰへ ﾊﾟﾚｯﾄ供給OK
      LDI     X0B1  ; (第一)搬送前進端
      ANI     X0B3  ; (第一)搬送中間端
      ORI     M1  ; 常時 OFF
      ANB
      ANI     X0B4  ; (第一)搬送異常
      OUT     L400  ; ﾄﾗﾝｻｰへ ﾊﾟﾚｯﾄ供給OK
11500 LD      M3001  ; ﾄﾗﾝｻｰへ ﾊﾟﾚｯﾄ供給
      OR      M3002  ; ﾄﾗﾝｻｰへ ﾊﾟﾚｯﾄ供給OK
      LDI     X0B1  ; (第一)搬送前進端
      ORI     M1  ; 常時 OFF
      ANB
      ANI     X0B4  ; (第一)搬送異常
      OUT     M3002  ; ﾄﾗﾝｻｰへ ﾊﾟﾚｯﾄ供給OK
11507 LD      T248  ; 下流ｽﾄｯﾊﾟｰﾊﾟﾚｯﾄ検出
      OR      M841  ; 下流ｽﾄｯﾊﾟｰﾊﾟﾚｯﾄ検出記憶
      LDI     M1  ; 常時 OFF
      AND     M3005  ; 工程完了補助
      ANI     X0B4  ; (第一)搬送異常
      ORB
      OUT     M3005  ; 工程完了補助
11514 LD      X265  ; ﾄﾗﾝｻｰﾊﾟﾚｯﾄ有り
      AND     M3003  ; 引込みﾌﾟｯｼｬｰ前進記憶
      AND     M847  ; 引込みﾌﾟｯｼｬｰ後退
      ANI     M318  ; 引込みﾌﾟｯｼｬｰ前進端
      OR      L200  ; ﾄﾗﾝｻｰﾊﾟﾚｯﾄ有り
      ANI     X0B1  ; (第一)搬送前進端
      OUT     L200  ; ﾄﾗﾝｻｰﾊﾟﾚｯﾄ有り
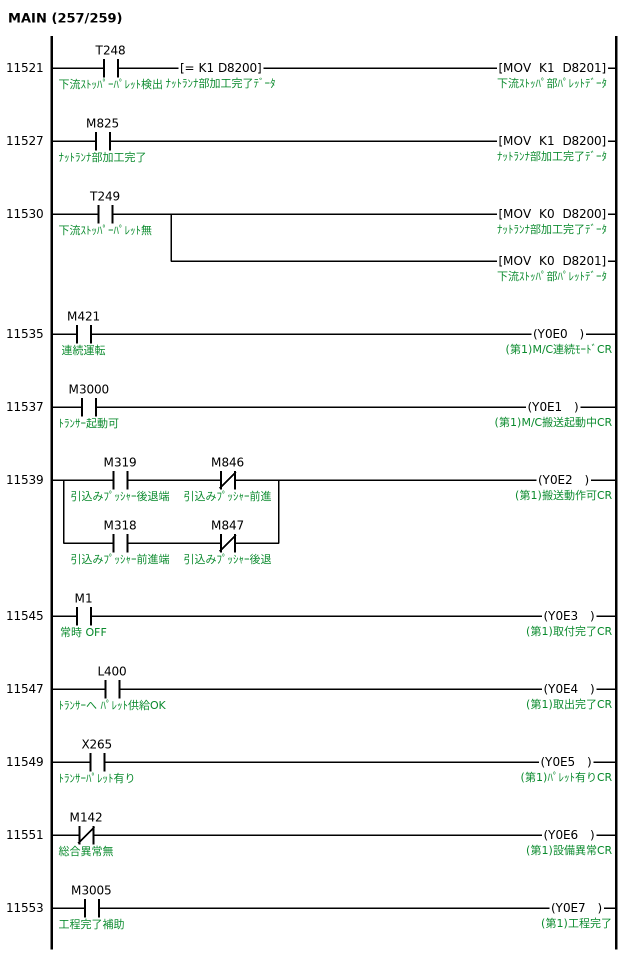
11521 LD      T248  ; 下流ｽﾄｯﾊﾟｰﾊﾟﾚｯﾄ検出
      AND=    K1 D8200  ; ﾅｯﾄﾗﾝﾅ部加工完了ﾃﾞｰﾀ
      MOV     K1 D8201  ; 下流ｽﾄｯﾊﾟ部ﾊﾟﾚｯﾄﾃﾞｰﾀ
11527 LD      M825  ; ﾅｯﾄﾗﾝﾅ部加工完了
      MOV     K1 D8200
11530 LD      T249  ; 下流ｽﾄｯﾊﾟｰﾊﾟﾚｯﾄ無
      MOV     K0 D8200
      MOV     K0 D8201
11535 LD      M421  ; 連続運転
      OUT     Y0E0  ; (第1)M/C連続ﾓｰﾄﾞCR
11537 LD      M3000  ; ﾄﾗﾝｻｰ起動可
      OUT     Y0E1  ; (第1)M/C搬送起動中CR
11539 LD      M319  ; 引込みﾌﾟｯｼｬｰ後退端
      ANI     M846  ; 引込みﾌﾟｯｼｬｰ前進
      LD      M318  ; 引込みﾌﾟｯｼｬｰ前進端
      ANI     M847  ; 引込みﾌﾟｯｼｬｰ後退
      ORB
      OUT     Y0E2  ; (第1)搬送動作可CR
11545 LD      M1  ; 常時 OFF
      OUT     Y0E3  ; (第1)取付完了CR
11547 LD      L400  ; ﾄﾗﾝｻｰへ ﾊﾟﾚｯﾄ供給OK
      OUT     Y0E4  ; (第1)取出完了CR
11549 LD      X265  ; ﾄﾗﾝｻｰﾊﾟﾚｯﾄ有り
      OUT     Y0E5  ; (第1)ﾊﾟﾚｯﾄ有りCR
11551 LDI     M142  ; 総合異常無
      OUT     Y0E6  ; (第1)設備異常CR
11553 LD      M3005  ; 工程完了補助
      OUT     Y0E7  ; (第1)工程完了
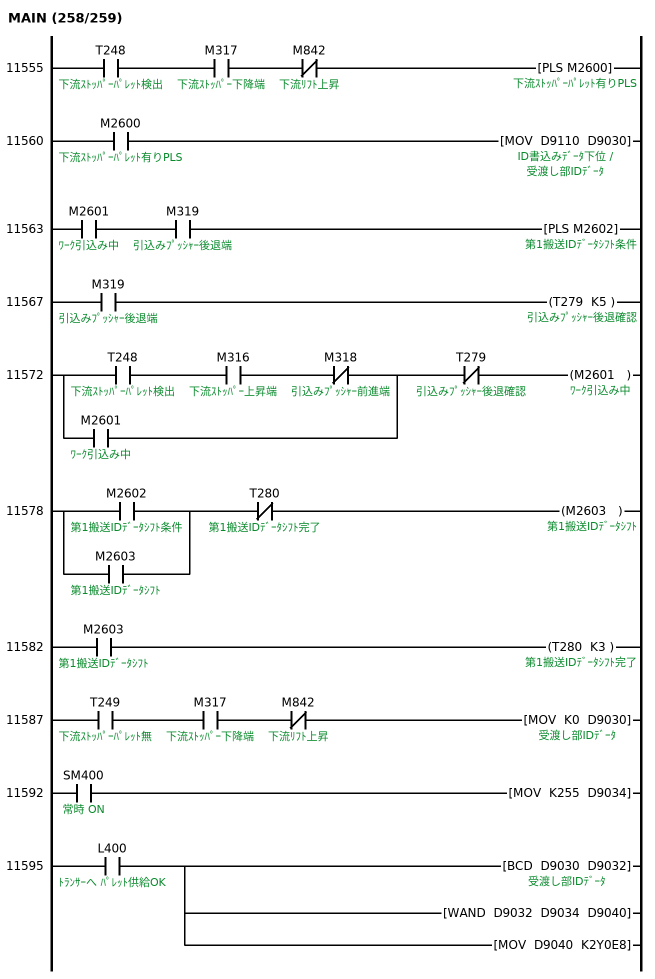
11555 LD      T248  ; 下流ｽﾄｯﾊﾟｰﾊﾟﾚｯﾄ検出
      AND     M317  ; 下流ｽﾄｯﾊﾟｰ下降端
      ANI     M842  ; 下流ﾘﾌﾄ上昇
      PLS     M2600  ; 下流ｽﾄｯﾊﾟｰﾊﾟﾚｯﾄ有りPLS
11560 LD      M2600  ; 下流ｽﾄｯﾊﾟｰﾊﾟﾚｯﾄ有りPLS
      MOV     D9110 D9030  ; 受渡し部IDﾃﾞｰﾀ
11563 LD      M2601  ; ﾜｰｸ引込み中
      AND     M319  ; 引込みﾌﾟｯｼｬｰ後退端
      PLS     M2602  ; 第1搬送IDﾃﾞｰﾀｼﾌﾄ条件
11567 LD      M319  ; 引込みﾌﾟｯｼｬｰ後退端
      OUT     T279 K5  ; 引込みﾌﾟｯｼｬｰ後退確認
11572 LD      T248  ; 下流ｽﾄｯﾊﾟｰﾊﾟﾚｯﾄ検出
      AND     M316  ; 下流ｽﾄｯﾊﾟｰ上昇端
      ANI     M318  ; 引込みﾌﾟｯｼｬｰ前進端
      OR      M2601  ; ﾜｰｸ引込み中
      ANI     T279  ; 引込みﾌﾟｯｼｬｰ後退確認
      OUT     M2601  ; ﾜｰｸ引込み中
11578 LD      M2602  ; 第1搬送IDﾃﾞｰﾀｼﾌﾄ条件
      OR      M2603  ; 第1搬送IDﾃﾞｰﾀｼﾌﾄ
      ANI     T280  ; 第1搬送IDﾃﾞｰﾀｼﾌﾄ完了
      OUT     M2603  ; 第1搬送IDﾃﾞｰﾀｼﾌﾄ
11582 LD      M2603  ; 第1搬送IDﾃﾞｰﾀｼﾌﾄ
      OUT     T280 K3  ; 第1搬送IDﾃﾞｰﾀｼﾌﾄ完了
11587 LD      T249  ; 下流ｽﾄｯﾊﾟｰﾊﾟﾚｯﾄ無
      AND     M317  ; 下流ｽﾄｯﾊﾟｰ下降端
      ANI     M842  ; 下流ﾘﾌﾄ上昇
      MOV     K0 D9030
11592 LD      SM400  ; 常時 ON
      MOV     K255 D9034
11595 LD      L400  ; ﾄﾗﾝｻｰへ ﾊﾟﾚｯﾄ供給OK
      BCD     D9030 D9032
      WAND    D9032 D9034 D9040
      MOV     D9040 K2Y0E8  ; (第1)ID情報 BCD 01 CR
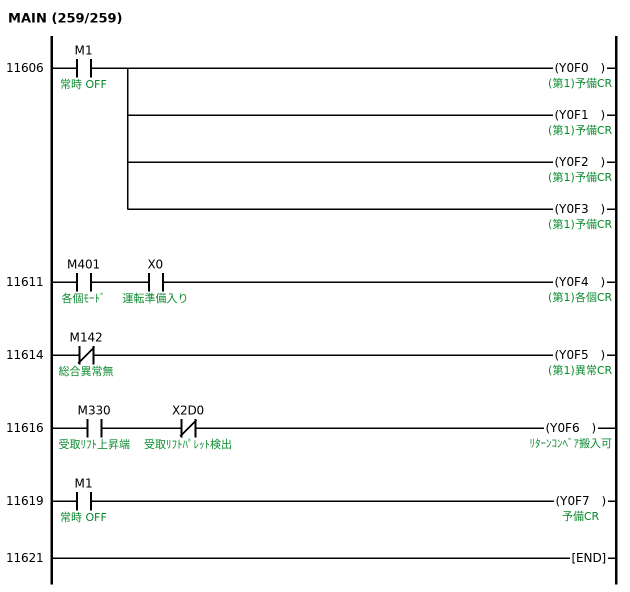
11606 LD      M1  ; 常時 OFF
      OUT     Y0F0  ; (第1)予備CR
      OUT     Y0F1  ; (第1)予備CR
      OUT     Y0F2  ; (第1)予備CR
      OUT     Y0F3  ; (第1)予備CR
11611 LD      M401  ; 各個ﾓｰﾄﾞ
      AND     X0  ; 運転準備入り
      OUT     Y0F4  ; (第1)各個CR
11614 LDI     M142  ; 総合異常無
      OUT     Y0F5  ; (第1)異常CR
11616 LD      M330  ; 受取ﾘﾌﾄ上昇端
      ANI     X2D0  ; 受取ﾘﾌﾄﾊﾟﾚｯﾄ検出
      OUT     Y0F6  ; ﾘﾀｰﾝｺﾝﾍﾞｱ搬入可
11619 LD      M1  ; 常時 OFF
      OUT     Y0F7  ; 予備CR
11621 END
END_PROGRAM

// device comments not shown above
M887  ; ﾛﾎﾞｯﾄﾌﾟﾛｸﾞﾗﾑNo.128
X0B5  ; (第一)予備
X0B7  ; (第一)予備
X171  ; (第1)異常ｺｰﾄﾞ2
X172  ; (第1)異常ｺｰﾄﾞ4
X173  ; (第1)異常ｺｰﾄﾞ8
X181  ; (第2)異常ｺｰﾄﾞ2
X182  ; (第2)異常ｺｰﾄﾞ4
X183  ; (第2)異常ｺｰﾄﾞ8
X1B1  ; ﾘｰﾄﾞﾃﾞｰﾀ出力ﾋﾞｯﾄ1(OD1)
X1B2  ; ﾘｰﾄﾞﾃﾞｰﾀ出力ﾋﾞｯﾄ2(OD2)
X1B3  ; ﾘｰﾄﾞﾃﾞｰﾀ出力ﾋﾞｯﾄ3(OD3)
X1B5  ; ﾘｰﾄﾞﾃﾞｰﾀ出力ﾋﾞｯﾄ5(OD5)
X1B6  ; ﾘｰﾄﾞﾃﾞｰﾀ出力ﾋﾞｯﾄ6(OD6)
X1B7  ; ﾘｰﾄﾞﾃﾞｰﾀ出力ﾋﾞｯﾄ7(OD7)
X30C  ; ロボット1ｻｲｸﾙ完了
X30F  ; ﾛﾎﾞｯﾄｺﾝﾃｨﾆｭｰ許可
X310  ; ﾛﾎﾞｯﾄ ｴﾗｰ  1
X311  ; ﾛﾎﾞｯﾄ ｴﾗｰ  2
X312  ; ﾛﾎﾞｯﾄ ｴﾗｰ  4
X313  ; ﾛﾎﾞｯﾄ ｴﾗｰ  8
X314  ; ﾛﾎﾞｯﾄ ｴﾗｰ 10
X315  ; ﾛﾎﾞｯﾄ ｴﾗｰ 20
X316  ; ﾛﾎﾞｯﾄ ｴﾗｰ 40
X317  ; ﾛﾎﾞｯﾄ ｴﾗｰ 80
X318  ; ﾛﾎﾞｯﾄ ｴﾗｰ100
X319  ; ﾛﾎﾞｯﾄ ｴﾗｰ200
X31A  ; ﾛﾎﾞｯﾄ ｴﾗｰ400
X31B  ; ﾛﾎﾞｯﾄ ｴﾗｰ800
X31C  ; ﾛﾎﾞｯﾄSSﾓｰﾄﾞ
X323  ; RB OUT803
X324  ; RB OUT804
X325  ; RB OUT805
X326  ; RB OUT806
X327  ; RB OUT807
X328  ; RB OUT808
X32A  ; RB OUT810
X32B  ; RB OUT811
X32C  ; RB OUT812
X32D  ; RB OUT813
X32E  ; RB OUT814
X32F  ; RB OUT815
X330  ; RB OUT816
X331  ; RB OUT817
X332  ; RB OUT818
X333  ; RB OUT819
X334  ; RB OUT820
X335  ; RB OUT821
X336  ; RB OUT822
X337  ; RB OUT823
X338  ; RB OUT824
X339  ; RB OUT825
X33A  ; RB OUT826
X33B  ; RB OUT827
X33C  ; RB OUT828
X33D  ; RB OUT829
X33E  ; RB OUT830
X33F  ; RB OUT831
X340  ; RB OUT832
X341  ; RB OUT833
X342  ; RB OUT834
X343  ; RB OUT835
X344  ; RB OUT836
X345  ; RB OUT837
X346  ; RB OUT838
X347  ; RB OUT839
X348  ; RB OUT840
X349  ; RB OUT841
X34A  ; RB OUT842
X34B  ; RB OUT843
X34C  ; RB OUT844
X34D  ; RB OUT845
X34E  ; RB OUT846
X34F  ; RB OUT847
X350  ; RB OUT848
X351  ; RB OUT849
X352  ; RB OUT850
X353  ; RB OUT851
X354  ; RB OUT852
X355  ; RB OUT853
X356  ; RB OUT854
X357  ; RB OUT855
X358  ; RB OUT856
X359  ; RB OUT857
X35A  ; RB OUT858
X35B  ; RB OUT859
X35C  ; RB OUT860
X35D  ; RB OUT861
X35E  ; RB OUT862
X35F  ; RB OUT863
X360  ; RB OUT864
X361  ; RB OUT865
X362  ; RB OUT866
X363  ; RB OUT867
X364  ; RB OUT868
X365  ; RB OUT869
X366  ; RB OUT870
X367  ; RB OUT871
X36E  ; RB OUT878
X36F  ; RB OUT879
X37A  ; ｴﾗｰ状態ﾌﾗｸﾞ
X37B  ; ﾘﾓｰﾄ局ﾚﾃﾞｨｰ
Y0E9  ; (第1)ID情報 BCD 02 CR
Y0EA  ; (第1)ID情報 BCD 04 CR
Y0EB  ; (第1)ID情報 BCD 08 CR
Y0EC  ; (第1)ID情報 BCD 10 CR
Y0ED  ; (第1)ID情報 BCD 20 CR
Y0EE  ; (第1)ID情報 BCD 40 CR
Y0EF  ; (第1)ID情報 BCD 80 CR
Y1C2  ; ﾗｲﾄﾃﾞｰﾀ入力ﾋﾞｯﾄ 1
Y1C3  ; ﾗｲﾄﾃﾞｰﾀ入力ﾋﾞｯﾄ 2
Y1C4  ; ﾗｲﾄﾃﾞｰﾀ入力ﾋﾞｯﾄ 3
Y1C6  ; ﾗｲﾄﾃﾞｰﾀ入力ﾋﾞｯﾄ 5
Y1C7  ; ﾗｲﾄﾃﾞｰﾀ入力ﾋﾞｯﾄ 6
Y1C8  ; ﾗｲﾄﾃﾞｰﾀ入力ﾋﾞｯﾄ 7
Y301  ; ﾛﾎﾞｯﾄｺﾝﾃｨﾆｭｰｽﾀｰﾄ
Y304  ; ﾛﾎﾞｯﾄ割込みｽﾀｰﾄ
Y318  ; RB IN536
Y319  ; RB IN537
Y31A  ; RB IN538
Y31B  ; RB IN539
Y31C  ; RB IN540
Y31D  ; RB IN541
Y31E  ; RB IN542
Y31F  ; RB IN543
Y32A  ; RB IN554
Y32B  ; RB IN555
Y32C  ; RB IN556
Y32D  ; RB IN557
Y32E  ; RB IN558
Y32F  ; RB IN559
Y336  ; RB IN566
Y337  ; RB IN567
Y346  ; RB IN582
Y347  ; RB IN583
Y34E  ; RB IN590
Y358  ; RB IN600
Y359  ; RB IN601
Y35A  ; RB IN602
Y35B  ; RB IN603
Y35C  ; RB IN604
Y35D  ; RB IN605
Y35E  ; RB IN606
Y35F  ; RB IN607
Y360  ; RB IN608
Y361  ; RB IN609
Y362  ; RB IN610
Y363  ; RB IN611
Y364  ; RB IN612
Y365  ; RB IN613
Y366  ; RB IN614
Y367  ; RB IN615
Y368  ; RB IN616
Y369  ; RB IN617
Y36A  ; RB IN618
Y36B  ; RB IN619
Y36C  ; RB IN620
Y36D  ; RB IN621
Y36E  ; RB IN622
Y36F  ; RB IN623
B5  ; 異常5
B6  ; 異常6
B7  ; 異常7
B0C  ; 異常12
B1C  ; 異常28
B1D  ; 異常29
B1E  ; 異常30
B1F  ; 異常31
B2C  ; 異常44
B2D  ; 異常45
B2E  ; 異常46
B2F  ; 異常47
B5C  ; 異常92
B5D  ; 異常93
B5E  ; 異常94
B5F  ; 異常95
B6C  ; 異常108
B6D  ; 異常109
B6E  ; 異常110
B6F  ; 異常111
B74  ; 異常116
B75  ; 異常117
B77  ; 異常119
B78  ; 異常120
B79  ; 異常121
B7A  ; 異常122
B7B  ; 異常123
B7C  ; 異常124
B7D  ; 異常125
B0A6  ; 異常166
B0A7  ; 異常167
B0A8  ; 異常168
B0A9  ; 異常169
B0AA  ; 異常170
B0AB  ; 異常171
B0BD  ; 異常189
B0BE  ; 異常190
B0BF  ; 異常191
B0CC  ; 異常204
B0CD  ; 異常205
B0CE  ; 異常206
B0CF  ; 異常207
B0D3  ; 異常211
B0D4  ; 異常212
B0D5  ; 異常213
B0D6  ; 異常214
B0D7  ; 異常215
B0D8  ; 異常216
B0D9  ; 異常217
B0DA  ; 異常218
B0DB  ; 異常219
B0DC  ; 異常220
B0DD  ; 異常221
B0DE  ; 異常222
B0DF  ; 異常223
B0EE  ; 異常238
B0EF  ; 異常239
B0F8  ; 異常248
B0F9  ; 異常249
T150  ; ﾛﾎﾞｯﾄ部ﾁｬｯｸ開端OFF
